FUNCTION "LGF_RandomRange_DInt" : DInt
TITLE = LGF_RandomRange_DInt
{ S7_Optimized_Access := 'TRUE' }
AUTHOR : Siemens_Digital_Industries
FAMILY : LGF
NAME : LGF_RandomRange_DInt
//This function generates a random value in defined limits with each call.
//The random number has the data type DInt in the specified range.
   VAR_INPUT
      minValue : DInt;   // Minimum value of the range of the random number - lower border
      maxValue : DInt;   // Maximum value of the range of the random number - upper border
   END_VAR

   VAR_OUTPUT
      error : Bool;   // FALSE: No error  TRUE: An error occurred during the execution of the FB
      status : Word;   // 16#0000-16#7FFF: Status of the FB  16#8000-16#FFFF: Error identification (see following Table)
      subfunctionStatus : Word;   // Status or return value of called FB's, FC's and system blocks
   END_VAR

   VAR_TEMP
      tempTime {InstructionName := 'DTL'; LibVersion := '1.0'} : DTL;   // Temp memory for System time
      tempNanoSecondInDWord : DWord;   // Temp UDInt converted to DWord for access to individual bytes
      tempTimeStatus : Word;   // Temp status of the instruction `RD_SYS_T`
      tempRandomValue : DWord;   // Temp Random startvalue
      tempNormReal : Real;   // Temp normalized Real value (0.0 - 1.0)
   END_VAR

   VAR CONSTANT
      ZERO : DInt := 0;   // Zero / 0.0 - value in case of  error
      MAX_UDINT : UDInt := 4294967295 ;   // Maximum DInt datatype
      SUB_STATUS_NO_ERROR : Word := 16#0000;   // Status: sub function call ends without error
      STATUS_FINISHED_NO_ERROR : Word := 16#0000;   // Execution finished without errors
      ERR_MAX_LESS_MIN : Word := 16#8200;   // Error: The ranges specified are wrong:  `minValue` is greater than `maxValue`
      ERR_RD_SYS_T : Word := 16#8600;   // Error in `RD_SYS_T` command - check `subFunctionStatus` code
   END_VAR


BEGIN
	REGION Block info header
	  //=============================================================================
	  // SIEMENS AG / (c)Copyright 2017
	  //-----------------------------------------------------------------------------
	  // Title:            LGF_RandomRange_DInt
	  // Comment/Function: This function generates random numbers in defined limits (Datatype DInt)
	  // Library/Family:   LGF(Library General Functions)
	  // Author:           Siemens Digital Industry Support
	  // Tested with:      S7-PLCSIM Advanced V2.0 SP1
	  // Engineering:      TIA Portal V15 Update 2
	  // Restrictions:     ENO disabled - error handling done by error and status
	  // Requirements:     PLC (S7-1200 / S7-1500)
	  //-------------------------------------------------------------------------------
	  // Change log table:
	  // Version  | Date       | Expert in charge       | Changes applied
	  //----------|------------|------------------------|------------------------------
	  // 01.00.00 19.08.2015  Siemens Industry Online Support
	  //                      First released version
	  // 01.00.01 02.01.2017  Siemens Industry Online Support
	  //                      Upgrade: TIA Portal V14 Update 1
	  // 01.00.02 17.08.2018  Siemens Industry Online Support
	  //                      Upgrade: TIA V15 Update 2
	  // 01.00.03 23.11.2018  Siemens Industry Online Support
	  //                      Upgrade: TIA V15.1
	  // 01.01.00 09.10.2019  Simatic Systems Support
	  //                      Renamed from "LGF_RandomInt" to "LGF_RandomRange_DInt"
	  //                      change random datatype from Int to DInt
	  //                      Regions, comments and constants are added
	  // 03.00.00 23.04.2020  Simatic Systems Support
	  //                      Set version to V3.0.0, harmonize the version of the whole library
	  // 03.00.01 04.02.2021  Simatic Systems Support
	  //                      Insert documentation
	  //=============================================================================
	END_REGION Block info header

	REGION DESCRIPTION
	  (/*
	Note
	:    The status of called commands is output in `subFunctionStatus`. In this case, the output value in `status` indicates which command caused the error. In this case, refer to the TIA Portal Online Help section for information on the respective commands.

	The block generates random values that are between the specified `minValue` and the `maxValue`. This random value is output via the `Ret_Val`.

	The random value is formed from the nanoseconds of the current system time of the CPU. The byte order of this value is inverted and then converted to a DInt.
	*/)
	END_REGION DESCRIPTION

	REGION Validation
	  // Check if the maximal Value is less than the minimal value
	  IF (#minValue > #maxValue) THEN
	    #error := true;
	    #status := #ERR_MAX_LESS_MIN;
	    #subfunctionStatus := #SUB_STATUS_NO_ERROR;
	    #LGF_RandomRange_DInt := #ZERO;
	    RETURN;
	  END_IF;

	  // Read system time
	  #tempTimeStatus := INT_TO_WORD(RD_SYS_T(#tempTime));

	  // Check return variable for error
	  IF (#tempTimeStatus <> #SUB_STATUS_NO_ERROR) THEN
	    #error := true;
	    #status := #ERR_RD_SYS_T;
	    #subfunctionStatus := #tempTimeStatus;
	    #LGF_RandomRange_DInt := #ZERO;
	    RETURN;
	  END_IF;
	END_REGION

	REGION Calculating random number
	  // Converting to double word so individual bytes can be addressed
	  #tempNanoSecondInDWord := UDINT_TO_DWORD(#tempTime.NANOSECOND);

	  // Callculate a random-start-value depending on the time
	  #tempRandomValue.%B3 := #tempNanoSecondInDWord.%B0;
	  #tempRandomValue.%B2 := #tempNanoSecondInDWord.%B1;
	  #tempRandomValue.%B1 := #tempNanoSecondInDWord.%B2;
	  #tempRandomValue.%B0 := #tempNanoSecondInDWord.%B3;

	  // Norm the calculated random number: 0.0 <= #tempNormReal <= 1.0
	  #tempNormReal := UDINT_TO_REAL(DWORD_TO_UDINT(#tempRandomValue)) / UDINT_TO_REAL(#MAX_UDINT);

	  // Scale the tempNormReal to be in the range of maxValue and minValue
	  #LGF_RandomRange_DInt := REAL_TO_DINT((#tempNormReal * DINT_TO_REAL(#maxValue - #minValue) + DINT_TO_REAL(#minValue)));

	  #error := false;
	  #status := #STATUS_FINISHED_NO_ERROR;
	  #subfunctionStatus := #SUB_STATUS_NO_ERROR;
	  // ENO mechanism is not used
	  ENO := TRUE;
	END_REGION

END_FUNCTION

